(* PLC project PLC, Beckhoff Automation GmbH TwinCAT PLC Control 3.5.13.21 *)
(* stored: creationDateTime 2024-02-17T22:43:16.3325174, modificationDateTime 2024-02-17T22:43:16.3325174 *)

TYPE PBResource :
STRUCT
	input: PBInput;
	config: PBConfig;
	status: PBStatus;
END_STRUCT
END_TYPE
